SUBAPPLICATION Uebung_210b (* Standard IEC 61131-3 FB_CTU (Vorwärtszähler, INT) mit Terminal-Ausgabe *)
  (* Standard: 61131-3; Description: Copyright (c) 2026 Meisterschulen am Ostbahnhof This program and the accompanying materials are made available under the terms of the Eclipse Public License 2.0 which is available at https://www.eclipse.org/legal/epl-2.0/ SPDX-License-Identifier: EPL-2.0 *)
  (* Version 1.1, 2026-04-21, Franz Höpfinger, Meisterschulen am Ostbahnhof, Added terminal output for counter value *)
  (* Version 1.0, 2026-04-20, Franz Höpfinger, Meisterschulen am Ostbahnhof, initial API and implementation (IEC 61131-3 version) *)
  PACKAGE Uebungen;
  IMPORT Uebungen::const::UT::DefaultPool_Numeric::OutputNumber_N3_N;
  IMPORT logiBUS::io::DI::logiBUS_DI::Input_I1;
  IMPORT logiBUS::io::DI::logiBUS_DI::Input_I2;
  IMPORT logiBUS::io::DQ::logiBUS_DO::Output_Q1;
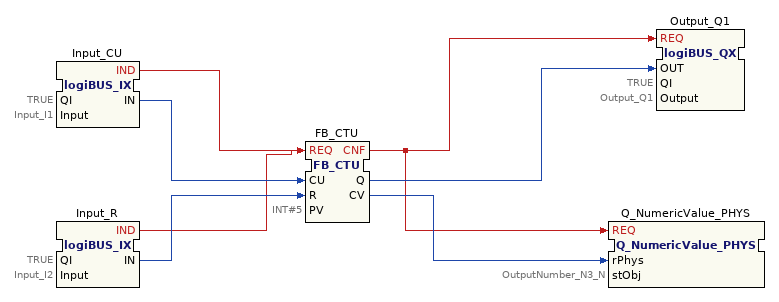
  (* F_INT_TO_UDINT ist großer Quatsch ... keine Negativen Zahlen möglich F_INT_TO_REAL kann man weglassen. jetzt geht auch negativ. z.B. PV auf INT#-5 *)
  (* hier gegebenenfalls einen E_D_FF einbauen, damit die Events reduziert werden. *)
  (* INT kann ohne Konvertierung auf REAL geschlossen werden. *)
  FBS
    FB_CTU : iec61131::counters::FB_CTU(PV := INT#5);
    Input_CU : logiBUS::io::DI::logiBUS_IX(QI := TRUE, Input := Input_I1);
    Input_R : logiBUS::io::DI::logiBUS_IX(QI := TRUE, Input := Input_I2);
    Output_Q1 : logiBUS::io::DQ::logiBUS_QX(QI := TRUE, Output := Output_Q1);
    Q_NumericValue_PHYS : isobus::UT::Q::Q_NumericValue_PHYS(stObj := OutputNumber_N3_N);
  END_FBS
  EVENT_CONNECTIONS
    Input_CU.IND TO FB_CTU.REQ;
    Input_R.IND TO FB_CTU.REQ;
    FB_CTU.CNF TO Output_Q1.REQ;
    FB_CTU.CNF TO Q_NumericValue_PHYS.REQ;
  END_CONNECTIONS
  DATA_CONNECTIONS
    Input_CU.IN TO FB_CTU.CU;
    Input_R.IN TO FB_CTU.R;
    FB_CTU.Q TO Output_Q1.OUT;
    FB_CTU.CV TO Q_NumericValue_PHYS.rPhys;
  END_CONNECTIONS
END_SUBAPPLICATION
